{attribute 'GeneratedUsingTerminal: CU2508-0000-0017'}
{attribute addProperty BoxType "CU2508-0000-0017"}
{attribute addProperty Id "EtcSlaveTerminalBaseEPM_Inputs_Channel_1AT %I*EPM_Inputs_Channel_385E794A2EPM_Inputs_Channel_2AT %I*EPM_Inputs_Channel_385E794A2EPM_Inputs_Channel_3AT %I*EPM_Inputs_Channel_385E794A2EPM_Inputs_Channel_4AT %I*EPM_Inputs_Channel_385E794A2EPM_Inputs_Channel_5AT %I*EPM_Inputs_Channel_385E794A2EPM_Inputs_Channel_6AT %I*EPM_Inputs_Channel_385E794A2EPM_Inputs_Channel_7AT %I*EPM_Inputs_Channel_385E794A2EPM_Inputs_Channel_8AT %I*EPM_Inputs_Channel_385E794A2EPM_Inputs_Channel_9AT %I*EPM_Inputs_Channel_385E794A2EPM_Inputs_Channel_10AT %I*EPM_Inputs_Channel_385E794A2WcStateAT %I*WcState_9091E0EB2InfoDataAT %I*InfoData_32EB74EA10"}
{attribute addProperty CRC "3356208334"}
{attribute addProperty Size "32"}
TYPE CU2508_C80BACCE EXTENDS EtcSlaveTerminalBase :
STRUCT
	{attribute addProperty Name "EPM_Inputs_Channel_1"}
	EPM_Inputs_Channel_1 : EPM_Inputs_Channel_385E794A;
	{attribute addProperty Name "EPM_Inputs_Channel_2"}
	EPM_Inputs_Channel_2 : EPM_Inputs_Channel_385E794A;
	{attribute addProperty Name "EPM_Inputs_Channel_3"}
	EPM_Inputs_Channel_3 : EPM_Inputs_Channel_385E794A;
	{attribute addProperty Name "EPM_Inputs_Channel_4"}
	EPM_Inputs_Channel_4 : EPM_Inputs_Channel_385E794A;
	{attribute addProperty Name "EPM_Inputs_Channel_5"}
	EPM_Inputs_Channel_5 : EPM_Inputs_Channel_385E794A;
	{attribute addProperty Name "EPM_Inputs_Channel_6"}
	EPM_Inputs_Channel_6 : EPM_Inputs_Channel_385E794A;
	{attribute addProperty Name "EPM_Inputs_Channel_7"}
	EPM_Inputs_Channel_7 : EPM_Inputs_Channel_385E794A;
	{attribute addProperty Name "EPM_Inputs_Channel_8"}
	EPM_Inputs_Channel_8 : EPM_Inputs_Channel_385E794A;
	{attribute addProperty Name "EPM_Inputs_Channel_9"}
	EPM_Inputs_Channel_9 : EPM_Inputs_Channel_385E794A;
	{attribute addProperty Name "EPM_Inputs_Channel_10"}
	EPM_Inputs_Channel_10 : EPM_Inputs_Channel_385E794A;
	{attribute addProperty Name "WcState"}
	WcState : WcState_9091E0EB;
	{attribute addProperty Name "InfoData"}
	InfoData : InfoData_32EB74EA;
END_STRUCT
END_TYPE

(* stored: Version 1.2.0.0, ProductVersion 3.1.4024.9
   DUT CU2508_C80BACCE: Id {27d8bdad-c9b9-442e-b012-ee1212e46e1c} *)
